// TIA Portal V20 export
TYPE "typeSequenceControlNodeHomeCheck_transferPnPLeft"
// stored: Namespace Unit1.Em5
   STRUCT
      waitPosPartNoDetect { ExternalWritable := 'False'} : Bool;
      waitPosPartDetect { ExternalWritable := 'False'} : Bool;
      sideTapePosPartNoDetect { ExternalWritable := 'False'} : Bool;
      sideTapePosPartDetect { ExternalWritable := 'False'} : Bool;
      hotPressLeftPosPartNoDetect { ExternalWritable := 'False'} : Bool;
      hotPressLeftPosPartDetect { ExternalWritable := 'False'} : Bool;
      hotPressRightPosPartNoDetect { ExternalWritable := 'False'} : Bool;
      hotPressRightPosPartDetect { ExternalWritable := 'False'} : Bool;
      hipotThicknessPosPartNoDetect { ExternalWritable := 'False'} : Bool;
      hipotThicknessPosPartDetect { ExternalWritable := 'False'} : Bool;
      defaultPosPartDetect : Bool;
      defaultPosPartNoDetect : Bool;
   END_STRUCT;
END_TYPE
